// TIA Portal V18 export
FUNCTION_BLOCK "_ML2_ts_block1_subunit"   // FB69, FBD
{ S7_Optimized_Access := 'TRUE' }
VERSION : 0.1
// stored: AutoNumber true, IsIECCheckEnabled false, IsRetainMemResEnabled false, MemoryReserve 100, SetENOAutomatically false, UDAEnableTagReadback false
   VAR_INPUT
      Q_mine : Int;
      Reset_all : Bool;
      CLK_flag : Bool;
   END_VAR
   VAR_OUTPUT
      P_flag : Bool;
      Q_flag : Bool;
   END_VAR
   VAR_IN_OUT
      Q_INT : Int;
   END_VAR
   VAR
      tr { S7_SetPoint := 'True'} : R_TRIG;
   END_VAR
BEGIN

REGION Network 1
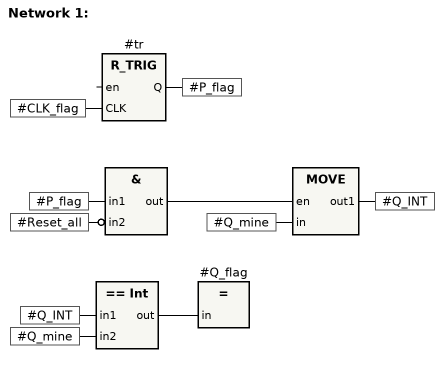
   #tr(CLK := #CLK_flag, Q => #P_flag);   // R_TRIG
   IF #P_flag AND NOT #Reset_all THEN #Q_INT := #Q_mine; END_IF;
   #Q_flag := #Q_INT = #Q_mine;
END_REGION
END_FUNCTION_BLOCK
